{attribute 'GeneratedUsingTerminal: EP7402-0057-0017'}
{attribute addProperty BoxType "EP7402-0057-0017"}
{attribute addProperty Id "OutputAT %Q*ARRAY[0..3] OF BOOL4Control_outputAT %Q*ARRAY[0..3] OF BOOL4"}
{attribute addProperty CRC "905683247"}
{attribute addProperty Size "8"}
TYPE DO_Outputs_A241BD3A EXTENDS OutputBase_10CEE7DE :
STRUCT
	{attribute addProperty Name "Output"}
	Output AT %Q* : ARRAY[0..3] OF BOOL;
	{attribute addProperty Name "Control_output"}
	Control_output AT %Q* : ARRAY[0..3] OF BOOL;
END_STRUCT
END_TYPE

(* stored: Version 1.2.0.0, ProductVersion 3.1.4024.11
   DUT DO_Outputs_A241BD3A: Id {4ebabc2b-dcdf-4b87-8d16-e8404c262cdb} *)
